(* CoDeSys 2.3.9.37 project: Cap12_5.pro *)
(* Libraries: Util.lib 18.5.10 16:14:28, standard.lib 4.10.05 12:14:46 *)

(* Global variable list: Global_Variables *)
VAR_GLOBAL
   (* Entradas *)
    IW1 : WORD;    (*Variable a controlar *)
   (* Entradas asociadas al panel de control *)
    ValorK : REAL:=1;
     ValorTN: REAL :=100;
     ValorTD:REAL :=0;
      ValorManual:BOOL:=FALSE;
     ValorSP:REAL:=1;
     ValorManualEnt:REAL:=1;

   (*Salidas*)
   QW1:WORD;    (*Actuación*)
END_VAR

(* POU PLC_PRG, ST *)
PROGRAM PLC_PRG
VAR
END_VAR
Proceso();
Control();
END_PROGRAM

(* POU Proceso, ST *)
PROGRAM Proceso
VAR
       K: REAL :=1;
       tau : REAL:=3000;
	tact: TIME;
	tactw: DWORD;
	tinc: REAL;
	toldw: DWORD;
	Salida: REAL;
	Entrada: REAL ;
       Ciclo1:BOOL:=TRUE;
	EscalaSalida: Escalado;
	IW1R: REAL;
	EscalaEntrada: Escalado;
	QW1R: REAL;
END_VAR
  QW1R:=WORD_TO_REAL(QW1);
  EscalaEntrada(Valor_Ent:=QW1R,Min_Ent:=0,Max_Ent:=4095,Min_Sal:=-10,Max_Sal:=10,Valor_Sal=>Entrada);

(* Programa que simula un sistema de primer orden *)
    tact:=TIME();
    tactw:=TIME_TO_DWORD(tact);
    (* Calcula el intervalo de tiempo desde el último ciclo en milisegundos *)
    tinc:=DWORD_TO_REAL(tactw-toldw);
    (* Almacena el valor actual para al próximo ciclo *)
    toldw:=tactw;
    IF Ciclo1=FALSE THEN
        Salida:=Salida+K*tinc*(Entrada-Salida)/tau;
    ELSE
        Ciclo1:=FALSE;
    END_IF

    EscalaSalida(Valor_Ent:=Salida,Min_Ent:=-10,Max_Ent:=10,Min_Sal:=0,Max_Sal:=4095,Valor_Sal=>IW1R);
    IW1:=REAL_TO_WORD(IW1R);
END_PROGRAM

(* POU Escalado, ST *)
FUNCTION_BLOCK Escalado
VAR_INPUT
	Valor_Ent : REAL;    (* Valor a convertir *)
	Min_Ent : REAL;      (* Valor mínimo de la entrada *)
	Max_Ent : REAL;	  (* Valor máximo de la entrada *)
	Min_Sal : REAL;      (* Valor mínimo de la salida *)
	Max_Sal : REAL;	   (* . Valor máximo de la salida. *)
       ValError : REAL:=-1;    (*Valor al que poner la salida en caso de error *)
END_VAR
VAR_OUTPUT
	Valor_Sal : REAL;   (*. Valor convertido *)
	Error :  BOOL;         (* Se activa cuando el valor de entrada queda fuera de límites *)
END_VAR
VAR
	pendiente: REAL;
END_VAR
Error:= (Valor_Ent>Max_Ent) OR (Valor_Ent<Min_Ent);

IF NOT Error THEN
   pendiente:=(Max_Sal-Min_Sal)/(Max_Ent-Min_Ent);
   Valor_Sal:=(Valor_Ent-Min_Ent)*pendiente+Min_Sal;
ELSE
   Valor_Sal:=ValError;
END_IF
END_FUNCTION_BLOCK

(* POU Control, FBD *)
PROGRAM Control
VAR
END_VAR
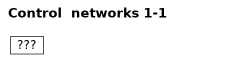
_FBD_ (* Function Block Diagram *)
NETWORK 1
	???
_END_FBD_
(* the same logic as Structured Text *)
(* Network 1 *)
END_PROGRAM

(* POU ControladorPI, ST *)
FUNCTION_BLOCK ControladorPI
VAR_INPUT
	Y :REAL;       (* Variable a controlar. *)
	SP : REAL;    (* Set Point, valor deseado de la variable a controlar.*)
	Kp : REAL := 1;     (* Parámetro del controlador. Proporcionar un valor por defecto de 1.0.*)
       TN : REAL:=1;       (* Parámetro del controlador *)
	Umin  : REAL :=0;   (* Valor mínimo de la salida. Por defecto tendrá el valor 0 *)
	UMax : REAL:=100;   (* Valor máximo de la salida. Por defecto, tendrá un valor 100.0.*)
	Offset :REAL:=0;     (* Cantidad a sumar a la señal del controlador. Por defecto tendrá un valor 0.*)
	Manual : BOOL;      (* TRUE modo manual, FALSE modo automático*)
	Manual_Ent : REAL;   (*Valor para la salida según ecuación (1.3) en modo manual *)
END_VAR
VAR_OUTPUT
	U : REAL;    (*Salida del controlador. *)
      Lim : BOOL;  (*Estará a TRUE si se superan los límites Umin o Umax en la salida *)
END_VAR
VAR
	tact: TIME;
	tactw: DWORD;
	tinc: REAL;
	toldw: DWORD;
	error: REAL;
	ierror: REAL;
      Ciclo1:BOOL :=TRUE;
END_VAR
   (* Calcula el instante de tiempo actual y se pasa a DWORD en milisegundos *)
    tact:=TIME();
    tactw:=TIME_TO_DWORD(tact);
    (* Calcula el intervalo de tiempo desde el último ciclo en milisegundos *)
    tinc:=DWORD_TO_REAL(tactw-toldw);
    (* Almacena el valor actual para al próximo ciclo *)
    toldw:=tactw;

IF Manual THEN
   U:=Manual_Ent+Offset;
   ierror:=0;
ELSE

    (* Calculo error ¨*)
   error:=SP-Y;
   (* Calculo de la integral del error  usando el método de Euler*)
   IF NOT Ciclo1 THEN
       ierror:=ierror+tinc*error;
  END_IF

   (* Calculo de la salida del conttrolador *)
  U:=Kp*(error+(1/TN)*ierror)+Offset;


END_IF


IF Ciclo1 THEN
   U:=Offset;
   Ciclo1:=FALSE;
END_IF


IF U>Umax THEN
     U:=Umax;
ELSE
   IF U<Umin THEN
       U:=Umin;
   END_IF
END_IF

LIM:=(U>Umax) OR  (U<Umin);
END_FUNCTION_BLOCK

(* Visualisation Visu
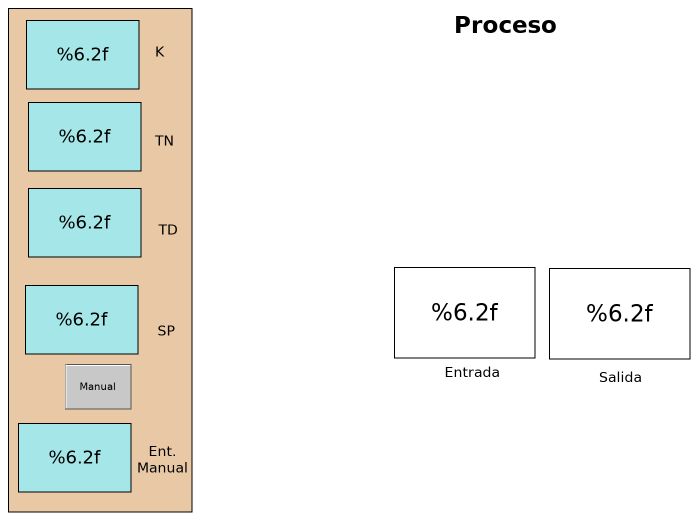
rectangle at (45,37)-(158,106): text "%6.2f"; shows ValorK; editable
rectangle at (129,43)-(228,94): text "K"
rectangle at (568,285)-(709,376): text "%6.2f"; shows Proceso.Salida
rectangle at (573,375)-(706,413): text "Salida"
rectangle at (44,302)-(157,371): text "%6.2f"; shows ValorSP; editable
rectangle at (136,322)-(235,373): text "SP"
button at (84,381)-(150,426): text "Manual"; toggles ValorManual
rectangle at (37,440)-(150,509): text "%6.2f"; shows ValorManualEnt; editable
rectangle at (458,23)-(591,61): text "Proceso"
rectangle at (413,284)-(554,375): text "%6.2f"; shows Proceso.Entrada
rectangle at (425,370)-(558,408): text "Entrada"
rectangle at (132,451)-(231,502): text "Ent. / Manual"
rectangle at (134,132)-(233,183): text "TN"
rectangle at (47,119)-(160,188): text "%6.2f"; shows ValorTN; editable
rectangle at (47,205)-(160,274): text "%6.2f"; shows ValorTD; editable
rectangle at (138,221)-(237,272): text "TD"
1 more shapes without text or variables
1 elements of other kinds (tables, trends, ...) not read
*)
